TYPE ST_VisuCtrlAxisFrame:
STRUCT
	sName				: string := 'Unknown';
	sUnit 				: STRING := 'Unknown';	(*  *)
	
	btnInit 			: BOOL;						(*  *)
	btnAbort 			: BOOL;						(*  *)
	btnReset			: BOOL;						(*  *)
	btnHome 			: BOOL;						(*  *)
	btnHalt				: BOOL;						(*  *)
	btnJogPositive 		: BOOL;						(*  *)
	btnJogNegative 		: BOOL;						(*  *)
	btnMoveTorque		: BOOL;
	btnMoveVelocity		: BOOL;
	btnMoveAbsolute		: BOOL;
	btnMoveAdditive		: BOOL;
	btnMoveRelative		: BOOL;
	btnStop				: BOOL;
	btnDecouple			: BOOL;
	btnCouple			: BOOL;
	btnUnLock			: BOOL;
	
	bActive				: BOOL;						(*  *)
	bHomed 				: BOOL;						(*  *)
	bInPosition 		: BOOL;						(*  *)
	bHalted				: BOOL;						(*  *)
	bError				: BOOL;						(*  *)
	iErrorID			: UDINT;					(*  *)
	
	lrActualPosition	: LREAL;					(*  *)
	lrActualVelocity	: LREAL;					(*  *)
	lrActualTorque		: LREAL;
	lrLagError			: LREAL;					(*  *)
	
	lrSetPosition		: LREAL;					(*  *)
	lrSetVelocity		: LREAL;					(*  *)
	lrSetTorque			: LREAL;
	
	lrOverride			: LREAL := 30.0;			(*  *)
	
	lrJogDistance 		: LREAL;					(*  *)
	lrJogVelocity		: LREAL;					(*  *)
	lrJogAcceleration	: LREAL;					(*  *)
	lrJogDeceleartion	: LREAL;					(*  *)
	
	sAxisImage			: STRING;					(*  *)
	eJogMode			: E_VisuCtrlAxisJogMode;	(*  *)
	eAxisState			: E_AxisState;				(*  *)
	sState				: STRING;					(* sState = ToString(eAxisState) *)
END_STRUCT
END_TYPE

(* stored: Version 1.1.0.1, ProductVersion 3.1.4024.12
   DUT ST_VisuCtrlAxisFrame: Id {c470a7f1-66bd-4257-be23-5042ae9ac889} *)
